{attribute 'TcGenerated'}
{attribute 'no-analysis'}
{attribute 'linkalways'}
// This function has been automatically generated from the project information.
VAR_GLOBAL CONSTANT
	{attribute 'const_non_replaced'}
	stLibVersion_XBoxControllerUtilities : ST_LibVersion := (iMajor := 1, iMinor := 0, iBuild := 0, iRevision := 0, nFlags := 1, sVersion := '1.0');
END_VAR

(* stored: Version 1.1.0.1, ProductVersion 3.1.4024.11
   GVL Global_Version: Id {581b72ee-e448-4281-95c0-0393a7284589} *)
